(* PLC project SafeLOGIC-1, BrAutomation SafeDESIGNER  4.3.4.4 *)
(* stored: companyURL http://www.br-automation.com, creationDateTime Fri Oct 19 13:14:02 2018 *)

PROGRAM Main

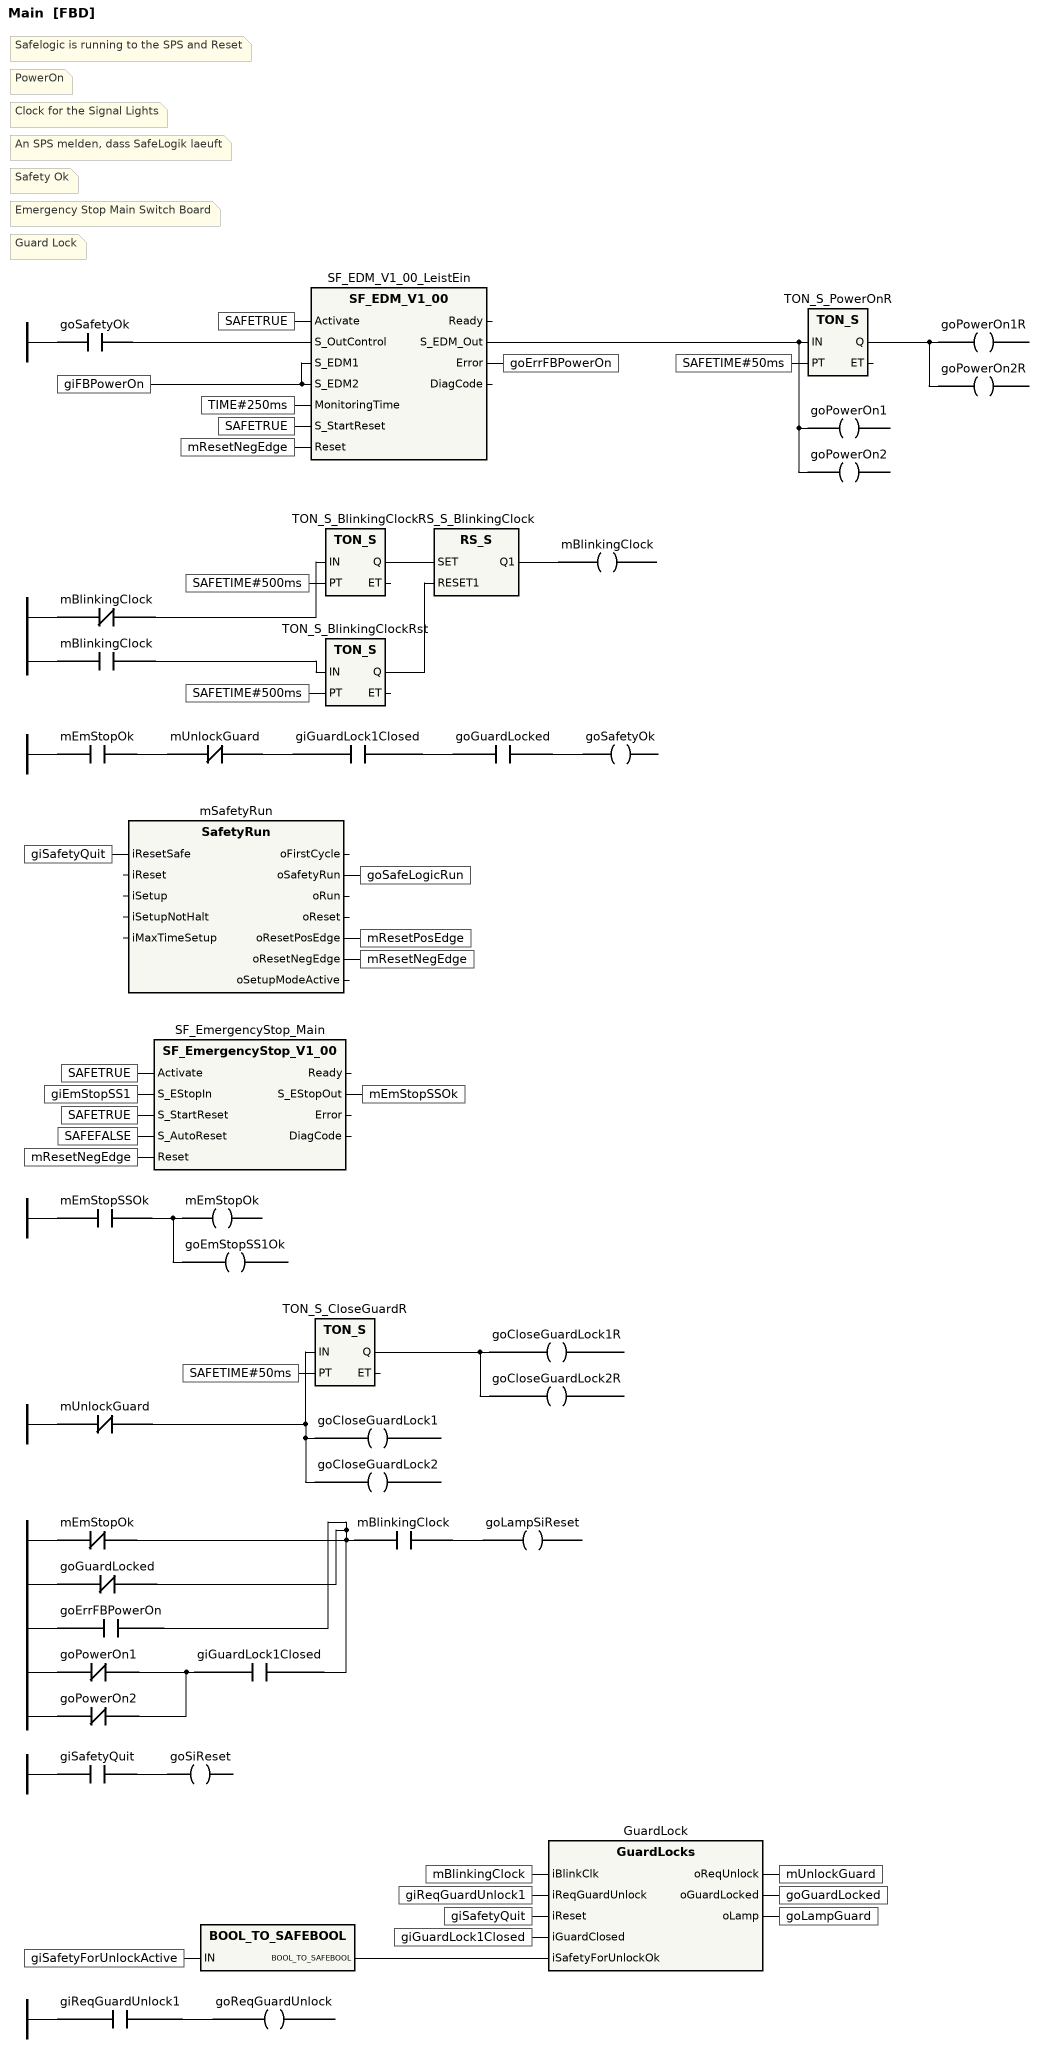
(* FBD diagram, written out as Structured Text *)
(* Safelogic is running to the SPS and Reset *)
(* An SPS melden, dass SafeLogik laeuft *)
mSafetyRun(iResetSafe := giSafetyQuit);
goSafeLogicRun := mSafetyRun.oSafetyRun;
mResetPosEdge := mSafetyRun.oResetPosEdge;
mResetNegEdge := mSafetyRun.oResetNegEdge;
(* Clock for the Signal Lights *)
TON_S_BlinkingClock(IN := NOT mBlinkingClock, PT := SAFETIME#500ms);
TON_S_BlinkingClockRst(IN := mBlinkingClock, PT := SAFETIME#500ms);
RS_S_BlinkingClock(SET := TON_S_BlinkingClock.Q, RESET1 := TON_S_BlinkingClockRst.Q);
mBlinkingClock := RS_S_BlinkingClock.Q1;
(* Emergency Stop Main Switch Board *)
SF_EmergencyStop_Main(Activate := SAFETRUE, S_EStopIn := giEmStopSS1, S_StartReset := SAFETRUE, S_AutoReset := SAFEFALSE, Reset := mResetNegEdge);
mEmStopSSOk := SF_EmergencyStop_Main.S_EStopOut;
mEmStopOk := mEmStopSSOk;
goEmStopSS1Ok := mEmStopSSOk;
(* Guard Lock *)
GuardLock(iBlinkClk := mBlinkingClock, iReqGuardUnlock := giReqGuardUnlock1, iReset := giSafetyQuit, iGuardClosed := giGuardLock1Closed, iSafetyForUnlockOk := BOOL_TO_SAFEBOOL(giSafetyForUnlockActive));
goLampGuard := GuardLock.oLamp;
mUnlockGuard := GuardLock.oReqUnlock;
goGuardLocked := GuardLock.oGuardLocked;
goReqGuardUnlock := giReqGuardUnlock1;
goCloseGuardLock1 := NOT mUnlockGuard;
goCloseGuardLock2 := NOT mUnlockGuard;
TON_S_CloseGuardR(IN := NOT mUnlockGuard, PT := SAFETIME#50ms);
goCloseGuardLock1R := TON_S_CloseGuardR.Q;
goCloseGuardLock2R := TON_S_CloseGuardR.Q;
(* Safety Ok *)
goSafetyOk := mEmStopOk AND NOT mUnlockGuard AND giGuardLock1Closed AND goGuardLocked;
(* PowerOn *)
SF_EDM_V1_00_LeistEin(Activate := SAFETRUE, S_OutControl := goSafetyOk, S_EDM1 := giFBPowerOn, S_EDM2 := giFBPowerOn, MonitoringTime := TIME#250ms, S_StartReset := SAFETRUE, Reset := mResetNegEdge);
goErrFBPowerOn := SF_EDM_V1_00_LeistEin.Error;
goPowerOn1 := SF_EDM_V1_00_LeistEin.S_EDM_Out;
TON_S_PowerOnR(IN := SF_EDM_V1_00_LeistEin.S_EDM_Out, PT := SAFETIME#50ms);
goPowerOn1R := TON_S_PowerOnR.Q;
goPowerOn2 := SF_EDM_V1_00_LeistEin.S_EDM_Out;
goPowerOn2R := TON_S_PowerOnR.Q;
goLampSiReset := (NOT mEmStopOk OR NOT goGuardLocked OR (NOT goPowerOn1 OR NOT goPowerOn2) AND giGuardLock1Closed OR goErrFBPowerOn) AND mBlinkingClock;
goSiReset := giSafetyQuit;
END_PROGRAM
